(* Logix 5000 project; controller BTS01 vendor 1 type 14 code 217 rev 32.14; software revision 32.04; part 5 of 15 *)
(* tags used below, declared in another part *)
   Alarm_Active : DINT;
   Alarm_TMR : TIMER[17,32];
   ALM_ENABLE : DINT[25];
   HMI_Global_Alarm_Ack_PB : BOOL;
   HMIAlarms : DINT[25];   // Alarm Trigger Array
   HMIAlarmsMsg : STRING64[17,32];   // Alarm Descriptions to Match Alarm Trigger Array
(* Alarm, continued *)

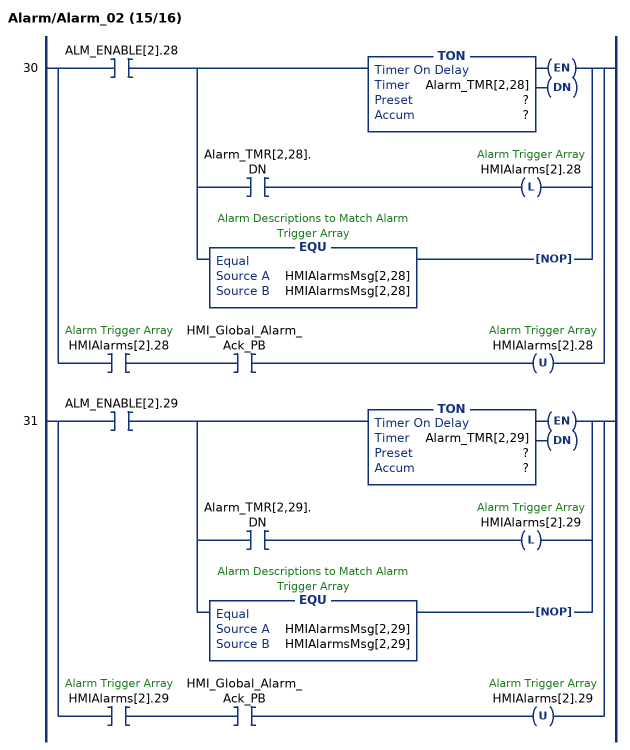
   [picture p69: Alarm/Alarm_02 rungs 30-31]
   30: [XIC(ALM_ENABLE[2].28) [TON(Alarm_TMR[2,28],?,?) ,XIC(Alarm_TMR[2,28].DN) OTL(HMIAlarms[2].28) ,EQU(HMIAlarmsMsg[2,28],HMIAlarmsMsg[2,28]) NOP() ] ,XIC(HMIAlarms[2].28) XIC(HMI_Global_Alarm_Ack_PB) OTU(HMIAlarms[2].28) ];
   31: [XIC(ALM_ENABLE[2].29) [TON(Alarm_TMR[2,29],?,?) ,XIC(Alarm_TMR[2,29].DN) OTL(HMIAlarms[2].29) ,EQU(HMIAlarmsMsg[2,29],HMIAlarmsMsg[2,29]) NOP() ] ,XIC(HMIAlarms[2].29) XIC(HMI_Global_Alarm_Ack_PB) OTU(HMIAlarms[2].29) ];
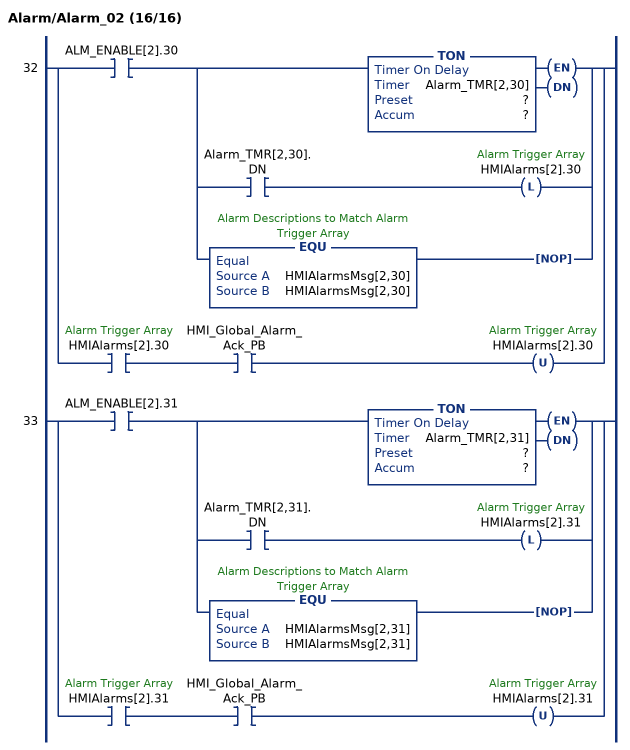
   32: [XIC(ALM_ENABLE[2].30) [TON(Alarm_TMR[2,30],?,?) ,XIC(Alarm_TMR[2,30].DN) OTL(HMIAlarms[2].30) ,EQU(HMIAlarmsMsg[2,30],HMIAlarmsMsg[2,30]) NOP() ] ,XIC(HMIAlarms[2].30) XIC(HMI_Global_Alarm_Ack_PB) OTU(HMIAlarms[2].30) ];
   33: [XIC(ALM_ENABLE[2].31) [TON(Alarm_TMR[2,31],?,?) ,XIC(Alarm_TMR[2,31].DN) OTL(HMIAlarms[2].31) ,EQU(HMIAlarmsMsg[2,31],HMIAlarmsMsg[2,31]) NOP() ] ,XIC(HMIAlarms[2].31) XIC(HMI_Global_Alarm_Ack_PB) OTU(HMIAlarms[2].31) ];
END_ROUTINE

ROUTINE Alarm_03   (* ladder *)
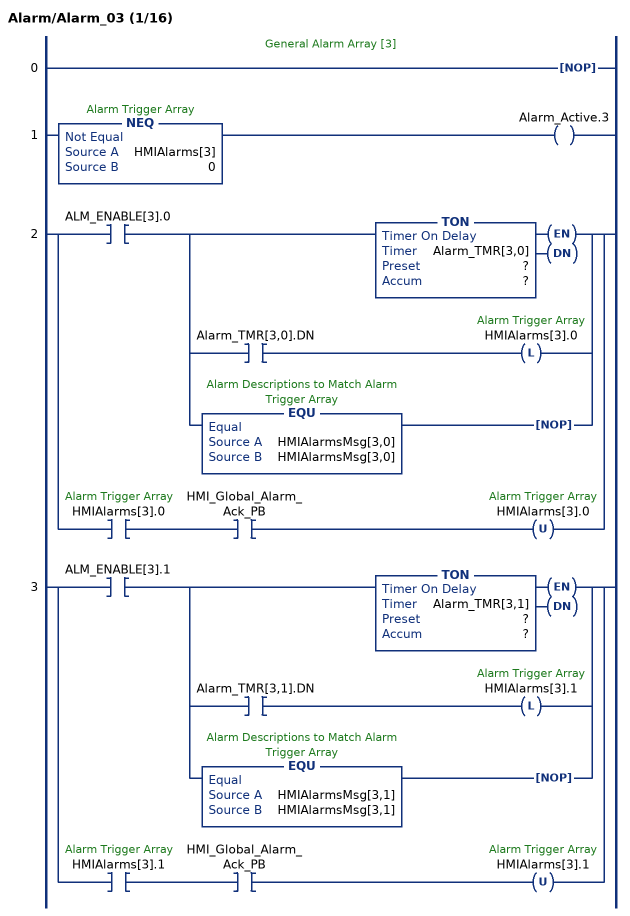
   // General Alarm Array [3]
   0: NOP();
   1: NEQ(HMIAlarms[3],0)OTE(Alarm_Active.3);
   2: [XIC(ALM_ENABLE[3].0) [TON(Alarm_TMR[3,0],?,?) ,XIC(Alarm_TMR[3,0].DN) OTL(HMIAlarms[3].0) ,EQU(HMIAlarmsMsg[3,0],HMIAlarmsMsg[3,0]) NOP() ] ,XIC(HMIAlarms[3].0) XIC(HMI_Global_Alarm_Ack_PB) OTU(HMIAlarms[3].0) ];
   3: [XIC(ALM_ENABLE[3].1) [TON(Alarm_TMR[3,1],?,?) ,XIC(Alarm_TMR[3,1].DN) OTL(HMIAlarms[3].1) ,EQU(HMIAlarmsMsg[3,1],HMIAlarmsMsg[3,1]) NOP() ] ,XIC(HMIAlarms[3].1) XIC(HMI_Global_Alarm_Ack_PB) OTU(HMIAlarms[3].1) ];
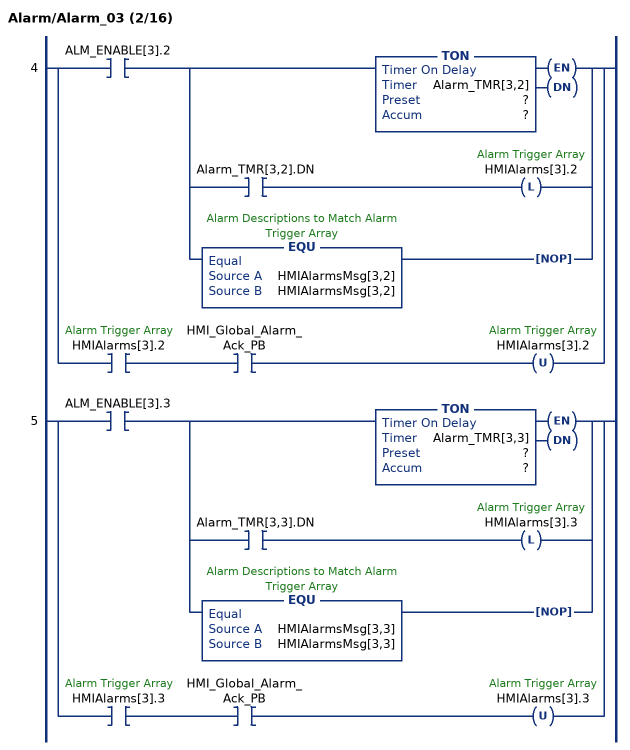
   4: [XIC(ALM_ENABLE[3].2) [TON(Alarm_TMR[3,2],?,?) ,XIC(Alarm_TMR[3,2].DN) OTL(HMIAlarms[3].2) ,EQU(HMIAlarmsMsg[3,2],HMIAlarmsMsg[3,2]) NOP() ] ,XIC(HMIAlarms[3].2) XIC(HMI_Global_Alarm_Ack_PB) OTU(HMIAlarms[3].2) ];
   5: [XIC(ALM_ENABLE[3].3) [TON(Alarm_TMR[3,3],?,?) ,XIC(Alarm_TMR[3,3].DN) OTL(HMIAlarms[3].3) ,EQU(HMIAlarmsMsg[3,3],HMIAlarmsMsg[3,3]) NOP() ] ,XIC(HMIAlarms[3].3) XIC(HMI_Global_Alarm_Ack_PB) OTU(HMIAlarms[3].3) ];
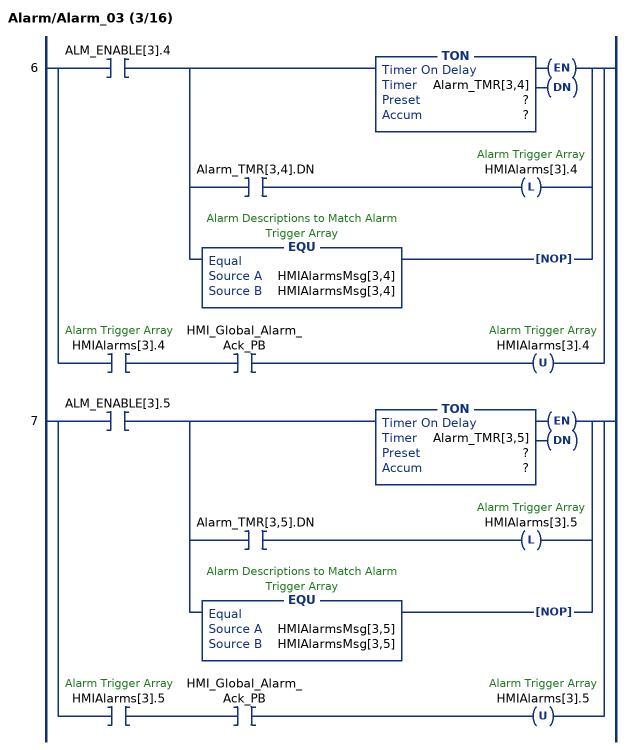
   6: [XIC(ALM_ENABLE[3].4) [TON(Alarm_TMR[3,4],?,?) ,XIC(Alarm_TMR[3,4].DN) OTL(HMIAlarms[3].4) ,EQU(HMIAlarmsMsg[3,4],HMIAlarmsMsg[3,4]) NOP() ] ,XIC(HMIAlarms[3].4) XIC(HMI_Global_Alarm_Ack_PB) OTU(HMIAlarms[3].4) ];
   7: [XIC(ALM_ENABLE[3].5) [TON(Alarm_TMR[3,5],?,?) ,XIC(Alarm_TMR[3,5].DN) OTL(HMIAlarms[3].5) ,EQU(HMIAlarmsMsg[3,5],HMIAlarmsMsg[3,5]) NOP() ] ,XIC(HMIAlarms[3].5) XIC(HMI_Global_Alarm_Ack_PB) OTU(HMIAlarms[3].5) ];
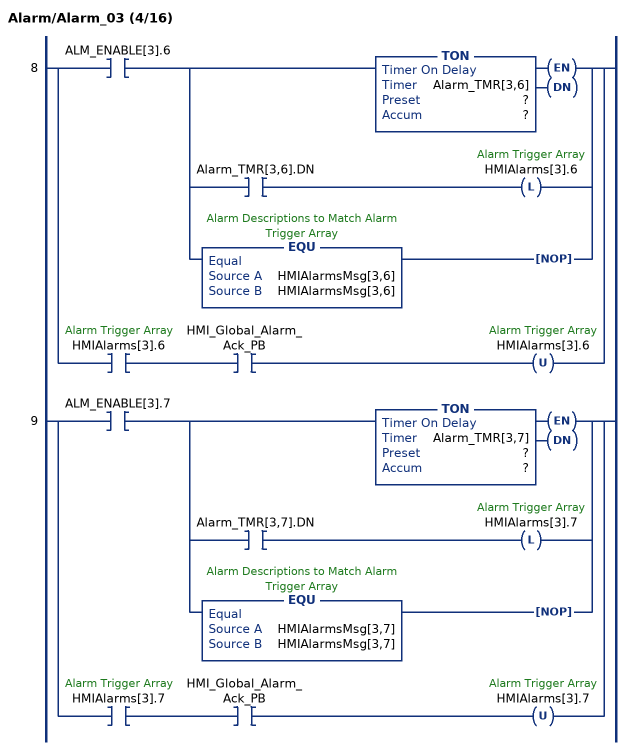
   8: [XIC(ALM_ENABLE[3].6) [TON(Alarm_TMR[3,6],?,?) ,XIC(Alarm_TMR[3,6].DN) OTL(HMIAlarms[3].6) ,EQU(HMIAlarmsMsg[3,6],HMIAlarmsMsg[3,6]) NOP() ] ,XIC(HMIAlarms[3].6) XIC(HMI_Global_Alarm_Ack_PB) OTU(HMIAlarms[3].6) ];
   9: [XIC(ALM_ENABLE[3].7) [TON(Alarm_TMR[3,7],?,?) ,XIC(Alarm_TMR[3,7].DN) OTL(HMIAlarms[3].7) ,EQU(HMIAlarmsMsg[3,7],HMIAlarmsMsg[3,7]) NOP() ] ,XIC(HMIAlarms[3].7) XIC(HMI_Global_Alarm_Ack_PB) OTU(HMIAlarms[3].7) ];
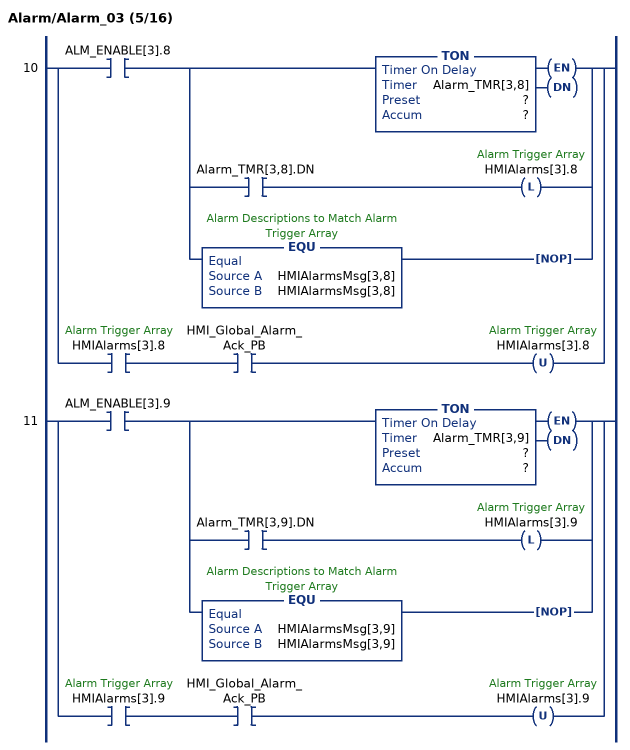
   10: [XIC(ALM_ENABLE[3].8) [TON(Alarm_TMR[3,8],?,?) ,XIC(Alarm_TMR[3,8].DN) OTL(HMIAlarms[3].8) ,EQU(HMIAlarmsMsg[3,8],HMIAlarmsMsg[3,8]) NOP() ] ,XIC(HMIAlarms[3].8) XIC(HMI_Global_Alarm_Ack_PB) OTU(HMIAlarms[3].8) ];
   11: [XIC(ALM_ENABLE[3].9) [TON(Alarm_TMR[3,9],?,?) ,XIC(Alarm_TMR[3,9].DN) OTL(HMIAlarms[3].9) ,EQU(HMIAlarmsMsg[3,9],HMIAlarmsMsg[3,9]) NOP() ] ,XIC(HMIAlarms[3].9) XIC(HMI_Global_Alarm_Ack_PB) OTU(HMIAlarms[3].9) ];
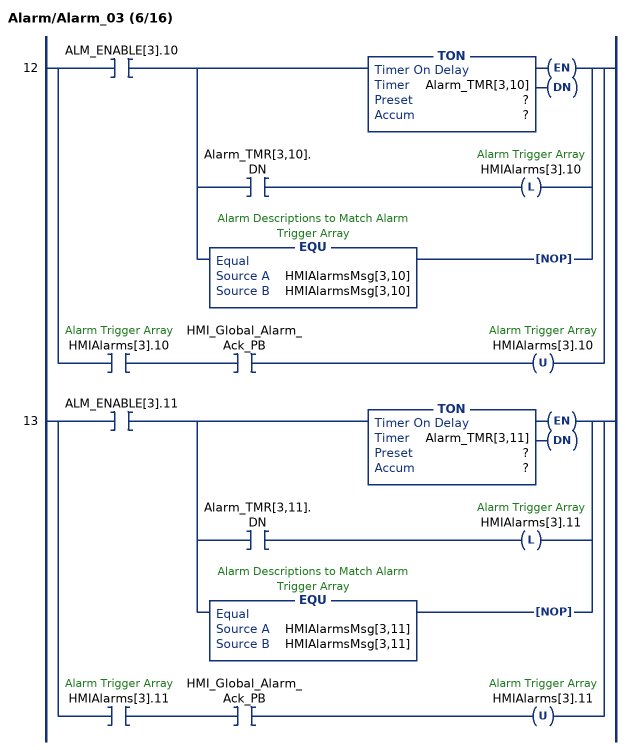
   12: [XIC(ALM_ENABLE[3].10) [TON(Alarm_TMR[3,10],?,?) ,XIC(Alarm_TMR[3,10].DN) OTL(HMIAlarms[3].10) ,EQU(HMIAlarmsMsg[3,10],HMIAlarmsMsg[3,10]) NOP() ] ,XIC(HMIAlarms[3].10) XIC(HMI_Global_Alarm_Ack_PB) OTU(HMIAlarms[3].10) ];
   13: [XIC(ALM_ENABLE[3].11) [TON(Alarm_TMR[3,11],?,?) ,XIC(Alarm_TMR[3,11].DN) OTL(HMIAlarms[3].11) ,EQU(HMIAlarmsMsg[3,11],HMIAlarmsMsg[3,11]) NOP() ] ,XIC(HMIAlarms[3].11) XIC(HMI_Global_Alarm_Ack_PB) OTU(HMIAlarms[3].11) ];
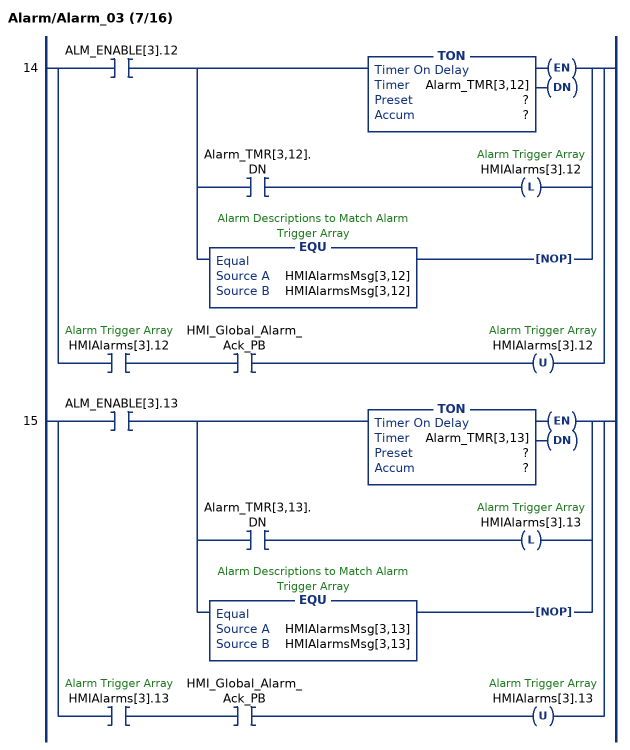
   14: [XIC(ALM_ENABLE[3].12) [TON(Alarm_TMR[3,12],?,?) ,XIC(Alarm_TMR[3,12].DN) OTL(HMIAlarms[3].12) ,EQU(HMIAlarmsMsg[3,12],HMIAlarmsMsg[3,12]) NOP() ] ,XIC(HMIAlarms[3].12) XIC(HMI_Global_Alarm_Ack_PB) OTU(HMIAlarms[3].12) ];
   15: [XIC(ALM_ENABLE[3].13) [TON(Alarm_TMR[3,13],?,?) ,XIC(Alarm_TMR[3,13].DN) OTL(HMIAlarms[3].13) ,EQU(HMIAlarmsMsg[3,13],HMIAlarmsMsg[3,13]) NOP() ] ,XIC(HMIAlarms[3].13) XIC(HMI_Global_Alarm_Ack_PB) OTU(HMIAlarms[3].13) ];
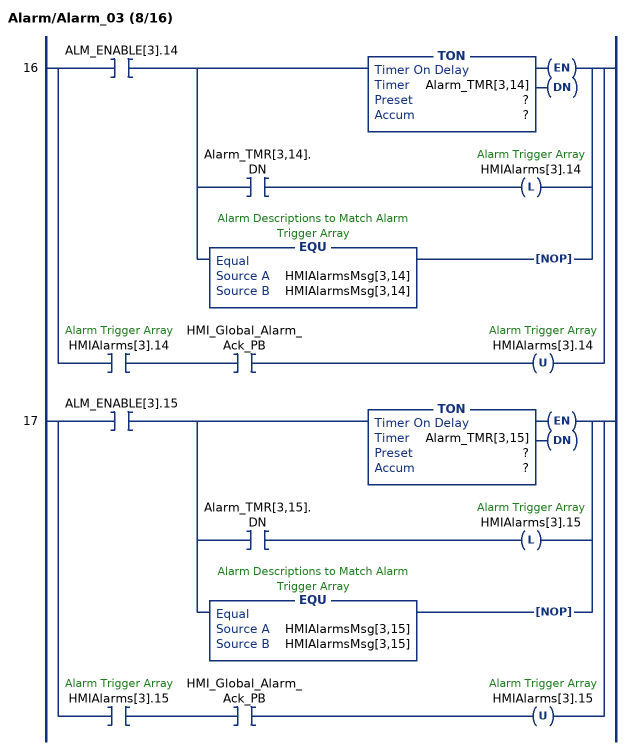
   16: [XIC(ALM_ENABLE[3].14) [TON(Alarm_TMR[3,14],?,?) ,XIC(Alarm_TMR[3,14].DN) OTL(HMIAlarms[3].14) ,EQU(HMIAlarmsMsg[3,14],HMIAlarmsMsg[3,14]) NOP() ] ,XIC(HMIAlarms[3].14) XIC(HMI_Global_Alarm_Ack_PB) OTU(HMIAlarms[3].14) ];
   17: [XIC(ALM_ENABLE[3].15) [TON(Alarm_TMR[3,15],?,?) ,XIC(Alarm_TMR[3,15].DN) OTL(HMIAlarms[3].15) ,EQU(HMIAlarmsMsg[3,15],HMIAlarmsMsg[3,15]) NOP() ] ,XIC(HMIAlarms[3].15) XIC(HMI_Global_Alarm_Ack_PB) OTU(HMIAlarms[3].15) ];
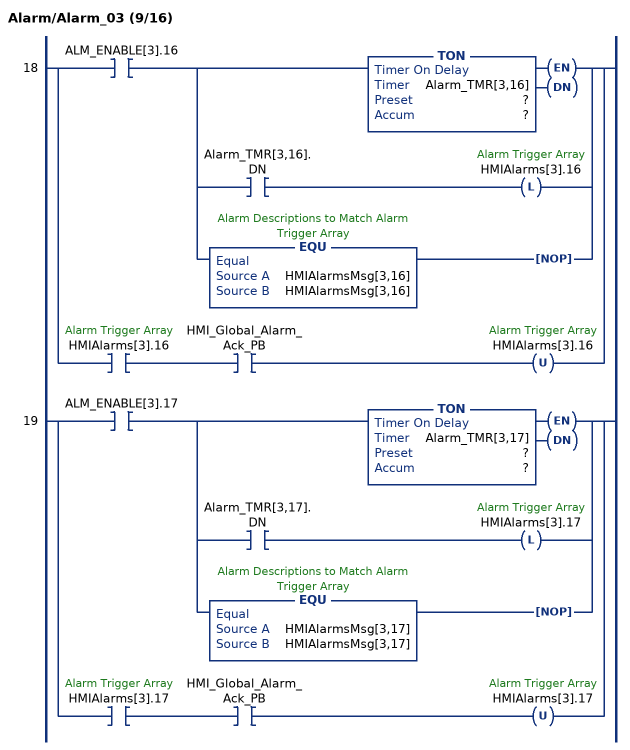
   18: [XIC(ALM_ENABLE[3].16) [TON(Alarm_TMR[3,16],?,?) ,XIC(Alarm_TMR[3,16].DN) OTL(HMIAlarms[3].16) ,EQU(HMIAlarmsMsg[3,16],HMIAlarmsMsg[3,16]) NOP() ] ,XIC(HMIAlarms[3].16) XIC(HMI_Global_Alarm_Ack_PB) OTU(HMIAlarms[3].16) ];
   19: [XIC(ALM_ENABLE[3].17) [TON(Alarm_TMR[3,17],?,?) ,XIC(Alarm_TMR[3,17].DN) OTL(HMIAlarms[3].17) ,EQU(HMIAlarmsMsg[3,17],HMIAlarmsMsg[3,17]) NOP() ] ,XIC(HMIAlarms[3].17) XIC(HMI_Global_Alarm_Ack_PB) OTU(HMIAlarms[3].17) ];
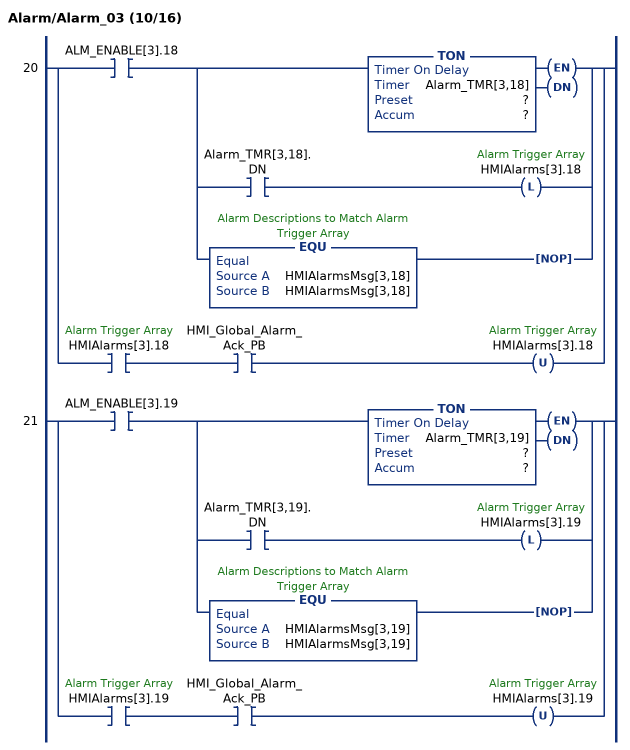
   20: [XIC(ALM_ENABLE[3].18) [TON(Alarm_TMR[3,18],?,?) ,XIC(Alarm_TMR[3,18].DN) OTL(HMIAlarms[3].18) ,EQU(HMIAlarmsMsg[3,18],HMIAlarmsMsg[3,18]) NOP() ] ,XIC(HMIAlarms[3].18) XIC(HMI_Global_Alarm_Ack_PB) OTU(HMIAlarms[3].18) ];
   21: [XIC(ALM_ENABLE[3].19) [TON(Alarm_TMR[3,19],?,?) ,XIC(Alarm_TMR[3,19].DN) OTL(HMIAlarms[3].19) ,EQU(HMIAlarmsMsg[3,19],HMIAlarmsMsg[3,19]) NOP() ] ,XIC(HMIAlarms[3].19) XIC(HMI_Global_Alarm_Ack_PB) OTU(HMIAlarms[3].19) ];
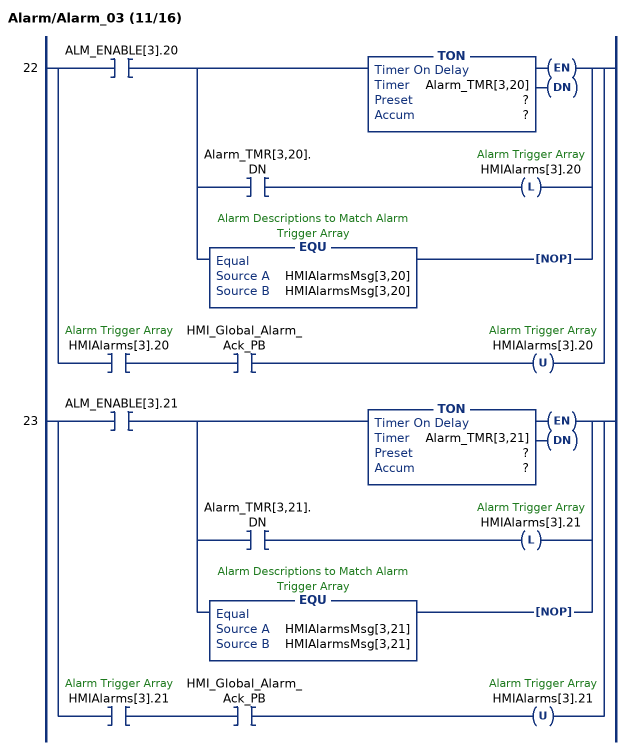
   22: [XIC(ALM_ENABLE[3].20) [TON(Alarm_TMR[3,20],?,?) ,XIC(Alarm_TMR[3,20].DN) OTL(HMIAlarms[3].20) ,EQU(HMIAlarmsMsg[3,20],HMIAlarmsMsg[3,20]) NOP() ] ,XIC(HMIAlarms[3].20) XIC(HMI_Global_Alarm_Ack_PB) OTU(HMIAlarms[3].20) ];
   23: [XIC(ALM_ENABLE[3].21) [TON(Alarm_TMR[3,21],?,?) ,XIC(Alarm_TMR[3,21].DN) OTL(HMIAlarms[3].21) ,EQU(HMIAlarmsMsg[3,21],HMIAlarmsMsg[3,21]) NOP() ] ,XIC(HMIAlarms[3].21) XIC(HMI_Global_Alarm_Ack_PB) OTU(HMIAlarms[3].21) ];
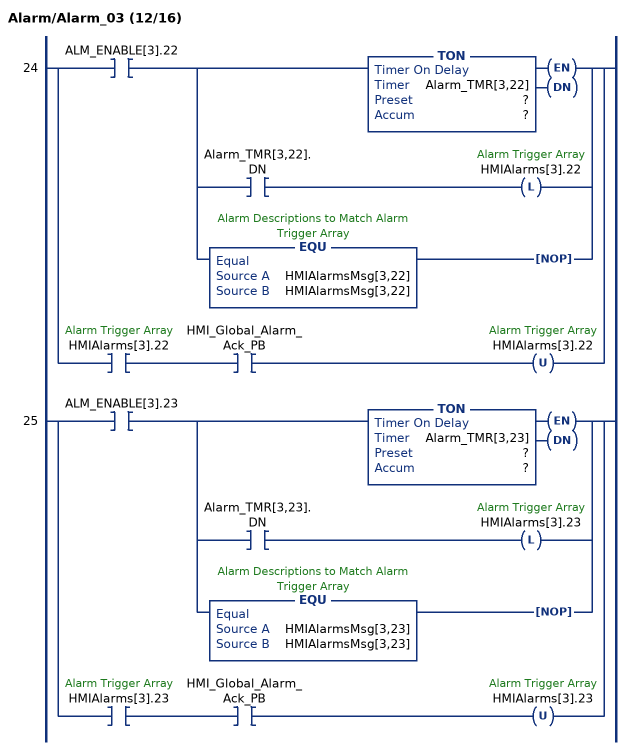
   24: [XIC(ALM_ENABLE[3].22) [TON(Alarm_TMR[3,22],?,?) ,XIC(Alarm_TMR[3,22].DN) OTL(HMIAlarms[3].22) ,EQU(HMIAlarmsMsg[3,22],HMIAlarmsMsg[3,22]) NOP() ] ,XIC(HMIAlarms[3].22) XIC(HMI_Global_Alarm_Ack_PB) OTU(HMIAlarms[3].22) ];
   25: [XIC(ALM_ENABLE[3].23) [TON(Alarm_TMR[3,23],?,?) ,XIC(Alarm_TMR[3,23].DN) OTL(HMIAlarms[3].23) ,EQU(HMIAlarmsMsg[3,23],HMIAlarmsMsg[3,23]) NOP() ] ,XIC(HMIAlarms[3].23) XIC(HMI_Global_Alarm_Ack_PB) OTU(HMIAlarms[3].23) ];
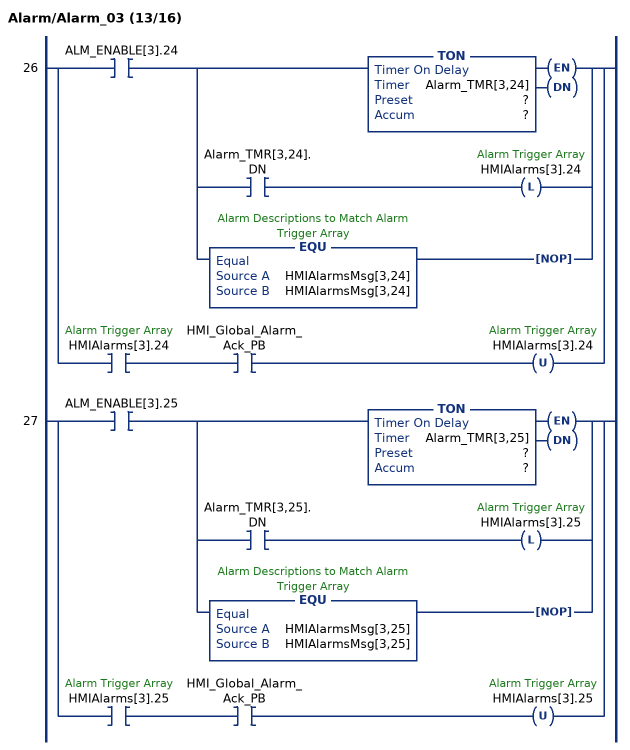
   26: [XIC(ALM_ENABLE[3].24) [TON(Alarm_TMR[3,24],?,?) ,XIC(Alarm_TMR[3,24].DN) OTL(HMIAlarms[3].24) ,EQU(HMIAlarmsMsg[3,24],HMIAlarmsMsg[3,24]) NOP() ] ,XIC(HMIAlarms[3].24) XIC(HMI_Global_Alarm_Ack_PB) OTU(HMIAlarms[3].24) ];
   27: [XIC(ALM_ENABLE[3].25) [TON(Alarm_TMR[3,25],?,?) ,XIC(Alarm_TMR[3,25].DN) OTL(HMIAlarms[3].25) ,EQU(HMIAlarmsMsg[3,25],HMIAlarmsMsg[3,25]) NOP() ] ,XIC(HMIAlarms[3].25) XIC(HMI_Global_Alarm_Ack_PB) OTU(HMIAlarms[3].25) ];
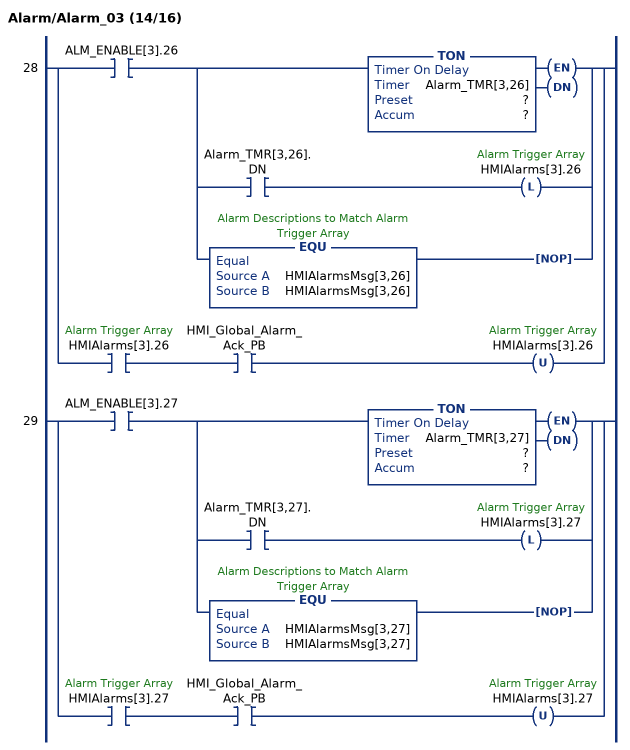
   28: [XIC(ALM_ENABLE[3].26) [TON(Alarm_TMR[3,26],?,?) ,XIC(Alarm_TMR[3,26].DN) OTL(HMIAlarms[3].26) ,EQU(HMIAlarmsMsg[3,26],HMIAlarmsMsg[3,26]) NOP() ] ,XIC(HMIAlarms[3].26) XIC(HMI_Global_Alarm_Ack_PB) OTU(HMIAlarms[3].26) ];
   29: [XIC(ALM_ENABLE[3].27) [TON(Alarm_TMR[3,27],?,?) ,XIC(Alarm_TMR[3,27].DN) OTL(HMIAlarms[3].27) ,EQU(HMIAlarmsMsg[3,27],HMIAlarmsMsg[3,27]) NOP() ] ,XIC(HMIAlarms[3].27) XIC(HMI_Global_Alarm_Ack_PB) OTU(HMIAlarms[3].27) ];
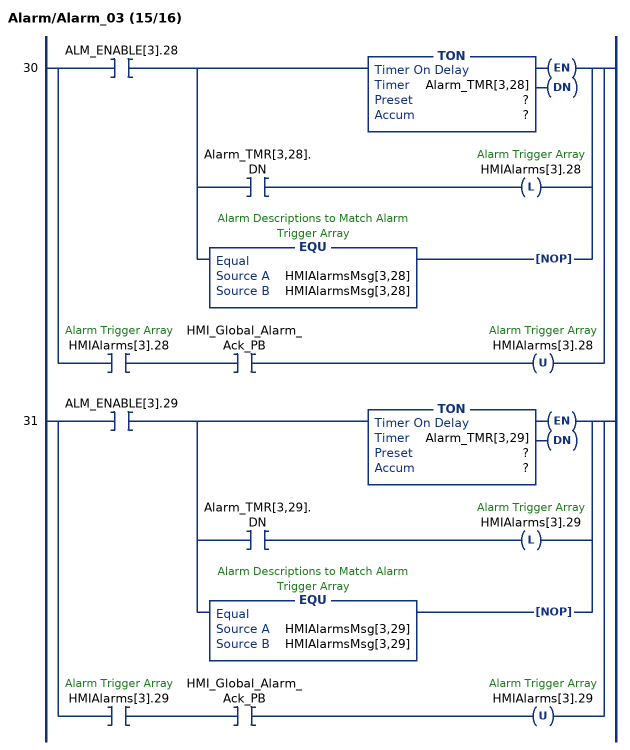
   30: [XIC(ALM_ENABLE[3].28) [TON(Alarm_TMR[3,28],?,?) ,XIC(Alarm_TMR[3,28].DN) OTL(HMIAlarms[3].28) ,EQU(HMIAlarmsMsg[3,28],HMIAlarmsMsg[3,28]) NOP() ] ,XIC(HMIAlarms[3].28) XIC(HMI_Global_Alarm_Ack_PB) OTU(HMIAlarms[3].28) ];
   31: [XIC(ALM_ENABLE[3].29) [TON(Alarm_TMR[3,29],?,?) ,XIC(Alarm_TMR[3,29].DN) OTL(HMIAlarms[3].29) ,EQU(HMIAlarmsMsg[3,29],HMIAlarmsMsg[3,29]) NOP() ] ,XIC(HMIAlarms[3].29) XIC(HMI_Global_Alarm_Ack_PB) OTU(HMIAlarms[3].29) ];
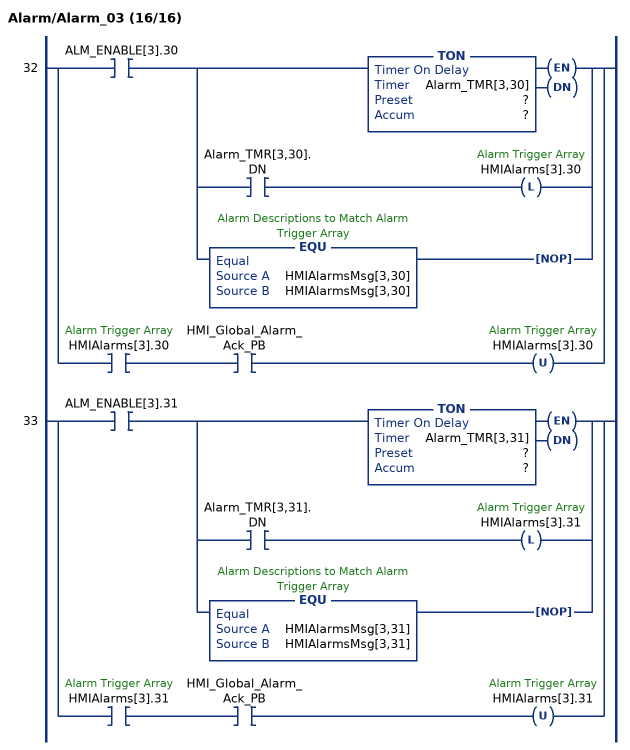
   32: [XIC(ALM_ENABLE[3].30) [TON(Alarm_TMR[3,30],?,?) ,XIC(Alarm_TMR[3,30].DN) OTL(HMIAlarms[3].30) ,EQU(HMIAlarmsMsg[3,30],HMIAlarmsMsg[3,30]) NOP() ] ,XIC(HMIAlarms[3].30) XIC(HMI_Global_Alarm_Ack_PB) OTU(HMIAlarms[3].30) ];
   33: [XIC(ALM_ENABLE[3].31) [TON(Alarm_TMR[3,31],?,?) ,XIC(Alarm_TMR[3,31].DN) OTL(HMIAlarms[3].31) ,EQU(HMIAlarmsMsg[3,31],HMIAlarmsMsg[3,31]) NOP() ] ,XIC(HMIAlarms[3].31) XIC(HMI_Global_Alarm_Ack_PB) OTU(HMIAlarms[3].31) ];
END_ROUTINE
